// TwinCAT 3 PLC project WorkshopLibrary
// Title: Workshop Library
// Company: BA Belgium
// Author: BA Belgium
// ProjectVersion: 1.0.0.0
// Description: Examples supplementary to the basic training
// ProgramVersion: 3.1.4026.20
// CompilerDefines: VISU_USEPROPERTYINFO
// libraries:
//   Tc2_Standard, * (Beckhoff Automation GmbH)
//   Tc2_System, * (Beckhoff Automation GmbH)
//   Tc3_Module, * (Beckhoff Automation GmbH)
// project tree:
//   Components/POUs/ LinTransfo.TcPOU
//   IO/POUs/ DigitalInputNC.TcPOU, DigitalInputNO.TcPOU, DigitalOutput.TcPOU, DigitalOutputLatched.TcPOU, MMotor.TcPOU, motoroef2_12.TcPOU, DigitalSwitch.TcPOU, DigitalSwitch4P.TcPOU
//   Project Information/ F_GetCompany.TcPOU, F_GetTitle.TcPOU, F_GetVersion.TcPOU
//   Templates/ _TemplateFB_1.TcPOU
//   Version/ Global_Version.TcGVL

// ---- Version/Global_Version.TcGVL
{attribute 'TcGenerated'}
{attribute 'no-analysis'}
{attribute 'linkalways'}
// This function has been automatically generated from the project information.
VAR_GLOBAL CONSTANT
	{attribute 'const_non_replaced'}
	stLibVersion_Workshop_Library : ST_LibVersion := (iMajor := 1, iMinor := 0, iBuild := 0, iRevision := 0, nFlags := 0, sVersion := '1.0.0.0');
END_VAR

// ---- Components/POUs/LinTransfo.TcPOU
FUNCTION_BLOCK LinTransfo
VAR_INPUT
	fIN				: REAL;
	fIN_min 		: REAL;
	fIN_max			: REAL;
	fOUT_min		: REAL;
	fOUT_max 		: REAL;
END_VAR
VAR_OUTPUT
	fOUT 			: REAL;	
END_VAR
VAR
END_VAR

fOUT := fOUT_min + (fIN - fIN_MIN) * (fOUT_max - fOUT_min) / (fIN_max - fIN_min);

END_FUNCTION_BLOCK

// ---- IO/POUs/DigitalInputNC.TcPOU
FUNCTION_BLOCK DigitalInputNC
VAR_INPUT
	input				: BOOL;
END_VAR
VAR_OUTPUT
	isActive			: BOOL;
	isNotActive			: BOOL;
	inputHasRisingEdge	: BOOL;
	inputHasFallingEdge	: BOOL;
END_VAR
VAR
	edgeR				: r_trig;
	edgeF				: f_trig;
END_VAR

isActive				:= NOT input;
isNotActive				:= input;

edgeR(CLK:=isActive, Q=>inputHasRisingEdge);
edgeF(CLK:=NOT isActive, Q=>inputHasFallingEdge);

END_FUNCTION_BLOCK

// ---- IO/POUs/DigitalInputNO.TcPOU
FUNCTION_BLOCK DigitalInputNO
VAR_INPUT
	input				: BOOL;
END_VAR
VAR_OUTPUT
	isActive			: BOOL;
	isNotActive			: BOOL;
	inputHasRisingEdge	: BOOL;
	inputHasFallingEdge	: BOOL;
END_VAR
VAR
	edgeR				: r_trig;
	edgeF				: f_trig;
END_VAR

isActive				:= input;
isNotActive				:= NOT input;

edgeR(CLK:=isActive, Q=>inputHasRisingEdge);
edgeF(CLK:=NOT isActive, Q=>inputHasFallingEdge);

END_FUNCTION_BLOCK

// ---- IO/POUs/DigitalOutput.TcPOU
FUNCTION_BLOCK DigitalOutput
VAR_INPUT
	on					: BOOL;
END_VAR
VAR_OUTPUT
	output				: BOOL;
END_VAR

output 					:= on;

END_FUNCTION_BLOCK

// ---- IO/POUs/DigitalOutputLatched.TcPOU
FUNCTION_BLOCK DigitalOutputLatched
VAR_INPUT
	on					: BOOL;
	off					: BOOL;
END_VAR
VAR_OUTPUT
	output				: BOOL;
END_VAR

IF off		THEN
	output 	:= FALSE;
ELSIF on 	THEN
	output 	:= TRUE;
END_IF

END_FUNCTION_BLOCK

// ---- IO/POUs/MMotor.TcPOU
FUNCTION_BLOCK MMotor
VAR_INPUT
	start AT %I* : BOOL;
	stop AT %I* : BOOL; 
END_VAR
VAR_OUTPUT
	motor AT %Q* : BOOL;
END_VAR
VAR
END_VAR

IF start THEN
	motor := TRUE;
ELSIF stop THEN
	motor := FALSE;
END_IF

END_FUNCTION_BLOCK

// ---- IO/POUs/motoroef2_12.TcPOU
FUNCTION_BLOCK motoroef2_12
VAR_INPUT
	DI_Inputsensorhoog : BOOL;
	DI_Inputsensorlaag : BOOL;
	DI_InputS1 			: BOOL;
	DI_InputS2			: BOOL;	
END_VAR
VAR_OUTPUT
	O_motordown 		: BOOL;
	O_motorup			: BOOL;
END_VAR
VAR
END_VAR



// Move UP: S2 pressed AND not at upper limit
IF DI_inputS2 AND NOT DI_inputsensorhoog THEN
    O_motorup := TRUE;
    O_motordown := FALSE;
END_IF

// Move DOWN: S1 pressed AND not at lower limit  
IF DI_inputS1 AND NOT DI_inputsensorlaag THEN
    O_motorup := FALSE;
    O_motordown := TRUE;
END_IF

// Safety: If both buttons pressed or at any limit, stop
IF (DI_inputS1 AND DI_inputS2) OR DI_inputsensorhoog OR DI_inputsensorlaag THEN
    O_motorup := FALSE;
    O_motordown := FALSE;
END_IF

END_FUNCTION_BLOCK

// ---- IO/POUs/DigitalSwitch.TcPOU
FUNCTION_BLOCK DigitalSwitch
VAR_INPUT
	input				: BOOL;
END_VAR
VAR_OUTPUT
	inPos00				: BOOL;
	inPos01				: BOOL;
END_VAR

inPos00 	:= NOT input;
inPos01		:= input;

END_FUNCTION_BLOCK

// ---- IO/POUs/DigitalSwitch4P.TcPOU
FUNCTION_BLOCK DigitalSwitch4P
VAR_INPUT
	input01				: BOOL;
	input02				: BOOL;
	input03				: BOOL;	
END_VAR
VAR_OUTPUT
	inPos00				: BOOL;
	inPos01				: BOOL;
	inPos02				: BOOL;
	inPos03				: BOOL;
END_VAR

inPos00		:= 
inPos01		:=
inPos02		:=
inPos03		:= FALSE;	

IF input01 		THEN
	inPos01		:= TRUE;	
ELSIF input02 	THEN
	inPos02		:= TRUE;	
ELSIF input03 	THEN
	inPos03		:= TRUE;	
ELSE
	inPos00		:= TRUE;	
END_IF

END_FUNCTION_BLOCK

// ---- Project Information/F_GetCompany.TcPOU
// This function has been automatically generated from the project information.
{attribute 'signature_flag' := '1073741824'}
{attribute 'TcGenerated'}
{attribute 'no-analysis'}
FUNCTION F_GetCompany : WSTRING
VAR_INPUT
	
END_VAR

F_GetCompany := "BA Belgium";

END_FUNCTION

// ---- Project Information/F_GetTitle.TcPOU
// This function has been automatically generated from the project information.
{attribute 'signature_flag' := '1073741824'}
{attribute 'TcGenerated'}
{attribute 'no-analysis'}
FUNCTION F_GetTitle : WSTRING
VAR_INPUT
	
END_VAR

F_GetTitle := "Workshop Library";

END_FUNCTION

// ---- Project Information/F_GetVersion.TcPOU
// This function has been automatically generated from the project information.
{attribute 'signature_flag' := '1073741824'}
{attribute 'TcGenerated'}
{attribute 'no-analysis'}
FUNCTION F_GetVersion : ST_LibVersion
VAR_INPUT
	
END_VAR

F_GetVersion.iMajor := 1;
F_GetVersion.iMinor := 0;
F_GetVersion.iBuild := 0;
F_GetVersion.iRevision := 0;
F_GetVersion.sVersion := '1.0.0.0';
F_GetVersion.nFlags := 0;

END_FUNCTION

// ---- Templates/_TemplateFB_1.TcPOU
{attribute 'no_explicit_call' := 'do not call this POU directly, call execute'} 
FUNCTION_BLOCK _TemplateFB_1
VAR
END_VAR

// NO CODE HERE, USE execute

METHOD execute
END_METHOD

END_FUNCTION_BLOCK
